FUNCTION Call_Emitter
VAR_INPUT
END_VAR
VAR
END_VAR

instEmitter(PartPresent:= BauteilVorEmitter, 
			CreatePart=> Emitter_Rollenband4m);
			
IF CreateNewPart THEN
	instEmitter.Create();
END_IF

IF BauteilVorEmitter THEN
	CreateNewPart := FALSE;
END_IF

END_FUNCTION

(* stored: Version 1.1.0.1
   POU Call_Emitter: Id {5eabb001-0730-44e4-adc3-7873d5c9fd23}, SpecialFunc None *)
